FUNCTION_BLOCK ABSTRACT PackMLModule EXTENDS Module IMPLEMENTS I_Module, I_ContainStatemachine
VAR
	_Statemachine : PackMLStatemachine_ModuleIntegrated('Statemachine');
	SequenceState : UDINT;
END_VAR

METHOD Aborted : BOOL;
Aborted := TRUE;
END_METHOD

METHOD Aborting : BOOL
Aborting := TRUE;
END_METHOD

METHOD Clearing : BOOL
Clearing := TRUE;
END_METHOD

METHOD Completed : BOOL
Completed := TRUE;
END_METHOD

METHOD Completing : BOOL
Completing := TRUE;
END_METHOD

METHOD CyclicLogic
StateSelect();
SUPER^.CyclicLogic();
END_METHOD

METHOD Execute : BOOL
Execute := TRUE;
END_METHOD

(*FB_Init is always available implicitly and it is used primarily for initialization.
The return value is not evaluated. For a specific influence, you can also declare the
methods explicitly and provide additional code there with the standard initialization
code. You can evaluate the return value.*)
METHOD FB_Init : BOOL
VAR_INPUT
	(* TRUE: the retain variables are initialized (reset warm / reset cold)*)
	bInitRetains	: BOOL;
	(* TRUE: the instance will be copied to the copy code afterward (online change)   *)
	bInCopyCode	: BOOL;
	Name	: T_MaxString;
END_VAR
_Statemachine.RegisterWithParent(THIS^);
END_METHOD

METHOD Held : BOOL
Held := TRUE;
END_METHOD

METHOD Holding : BOOL
Holding := TRUE;
END_METHOD

METHOD Idle : BOOL
Idle := TRUE;
END_METHOD

METHOD Resetting : BOOL
Resetting := TRUE;
END_METHOD

METHOD Starting : BOOL
Starting := TRUE;
END_METHOD

PROPERTY Statemachine : I_Statemachine
GET
Statemachine := _Statemachine;
END_GET
END_PROPERTY

METHOD PRIVATE StateSelect
VAR_INST
	ClearingTon : TON;
	LastState	: DINT;
END_VAR
IF LastState <> _Statemachine.CurrentState THEN
	SequenceState := 0;
	LastState	  := _Statemachine.CurrentState;
END_IF

CASE _Statemachine.CurrentState OF
	E_PMLState.Undefined:
		;

	E_PMLState.Clearing:
		ClearingTon(IN := TRUE, PT := ApplicationBaseParameter.ClearingTimeout);
		IF Clearing() THEN
			ClearingTon(IN := FALSE);
			_Statemachine.StateComplete();
		END_IF

		IF ClearingTon.Q THEN
			ClearingTon(IN := FALSE);
			Trace.LogMessage('Clearing Timeout exeeded! - ', _Name);
			_Statemachine.ChangeState(E_PMLCommand.Abort);
		END_IF

	E_PMLState.Stopped:
		Stopped();

	E_PMLState.Starting:
		IF Starting() THEN
			_Statemachine.StateComplete();
		END_IF

	E_PMLState.Idle:
		Idle();

	E_PMLState.Suspended:
		Suspended();

	E_PMLState.Execute:
		Execute();

	E_PMLState.Stopping:
		IF Stopping() THEN
			_Statemachine.StateComplete();
		END_IF

	E_PMLState.Aborting:
		IF Aborting() THEN
			_Statemachine.StateComplete();
		END_IF

	E_PMLState.Aborted:
		Aborted();

	E_PMLState.Holding:
		IF Holding() THEN
			_Statemachine.StateComplete();
		END_IF

	E_PMLState.Held:
		Held();

	E_PMLState.Unholding:
		IF Unholding() THEN
			_Statemachine.StateComplete();
		END_IF

	E_PMLState.Suspending:
		IF Suspending() THEN
			_Statemachine.StateComplete();
		END_IF

	E_PMLState.Unsuspending:
		IF Unsuspending() THEN
			_Statemachine.StateComplete();
		END_IF

	E_PMLState.Resetting:
		IF Resetting() THEN
			_Statemachine.StateComplete();
		END_IF

	E_PMLState.Completing:
		IF Completing() THEN
			_Statemachine.StateComplete();
		END_IF

	E_PMLState.Completed:
		Completed();
END_CASE
END_METHOD

METHOD Stopped : BOOL
Stopped := TRUE;
END_METHOD

METHOD Stopping : BOOL
Stopping := TRUE;
END_METHOD

METHOD Suspended : BOOL
Suspended := TRUE;
END_METHOD

METHOD Suspending : BOOL
Suspending := TRUE;
END_METHOD

METHOD Unholding : BOOL
Unholding := TRUE;
END_METHOD

METHOD Unsuspending : BOOL
Unsuspending := TRUE;
END_METHOD

END_FUNCTION_BLOCK

(* stored: Version 1.1.0.1, ProductVersion 3.1.4026.18
   POU PackMLModule: Id {25a20bd0-0f0a-4e0a-b97f-d7939b271cdf}, SpecialFunc None
   Folder Constructor: Id {a13ca037-f942-467a-ab9a-88458af13ff4}
   Folder States: Id {30dc58e5-9c9d-4518-aef5-bd9689273556}
   Method Aborted: Id {51e43f5d-fd8d-494c-8a5f-ea0bc5c40c2a}
   Method Aborting: Id {c4250865-8cbe-4aac-bcb8-82d7f21aeaa5}
   Method Clearing: Id {760bbabd-d445-48de-b531-bbeee9be9437}
   Method Completed: Id {373682f7-a515-4ca4-8760-e2da7bbf8afe}
   Method Completing: Id {5b6dc54d-dc43-4eaf-8acf-95ceb1c0e00f}
   Method CyclicLogic: Id {216b4710-59af-4382-82b8-ab4bd823dd52}
   Method Execute: Id {86dedc2b-a9d0-42ca-95c3-86d96e011557}
   Method FB_Init: Id {abcb1884-2b9f-44e1-bb9f-0b5403670a97}
   Method Held: Id {c57f029c-75c4-4ea1-a37e-b958c3da9f88}
   Method Holding: Id {34146d9f-8c3e-406e-b106-fa0ea7a05843}
   Method Idle: Id {40c63394-b723-48fe-993e-580bdd7b830f}
   Method Resetting: Id {bfc50916-07ee-49a4-813e-d83c1d593e36}
   Method Starting: Id {6cee2754-c5ab-4342-903e-29a875c97e85}
   Property Statemachine: Id {1c470240-50cc-47d0-b4e1-938f2e4bae3b}
   Get Get: Id {fcea9f8e-87e4-4500-b028-2bb2188b6a76}
   Method StateSelect: Id {13881525-b521-4102-aead-d8a7122bf0de}
   Method Stopped: Id {99231bb4-7b08-4edb-b042-bf5687beabf4}
   Method Stopping: Id {f408c09b-22f1-4812-801b-bbd5e5ec9b5e}
   Method Suspended: Id {770afc9d-016b-4468-9a81-323635dbafe6}
   Method Suspending: Id {6d800758-6d66-4ce6-ad6f-98ac21133cf4}
   Method Unholding: Id {8573ee61-26a5-47b0-ae1f-e16547c62787}
   Method Unsuspending: Id {d5a0cf5b-153b-4f83-b120-76ab413a17e1} *)
